TYPE ST_TEMP1_Save :
STRUCT
	id: DINT;
	timestamp: DT;
	temp1: STRING(45);
END_STRUCT
END_TYPE

(* stored: Version 1.1.0.1, ProductVersion 3.1.4018.5
   DUT ST_TEMP1_Save: Id {71441d62-68b9-4330-8069-14e50e275baa} *)
